Staubli VAL3: onF7Event.pgx

program onF7Event(bool& x_bSave[] (dimensions=1))
  local TrajectoryItem l_tTraj
  local num l_nItem
begin
  // look if the bButton is enable
  if bButton[6]
    //
    // insert
    l_nItem=nIndexItem
    // insert the default value
    call trajType:insertItem(nIndexItem,nIndexItem+1)
    call trajType:getTrajItem(l_tTraj,nIndexItem)
    l_tTraj.comment=""
    l_tTraj.toStop=false
    call trajType:setTrajItem(l_tTraj,nIndexItem+1)
    nIndexItem=nIndexItem+1
    // rebuild list
    call buildList()
    x_bSave=true
    //refresh
    call buildList()
    use:bUseRefresh=true
  endIf
end
